FUNCTION_BLOCK GEOLOC_SUBSCRIBER_SINGLE
  {SET_ATTRIBUTE(OpcUa, SERVICE)}
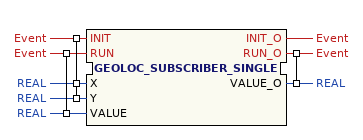
  EVENT_INPUT
    INIT WITH X, Y; (* FB Initialization *)
    RUN WITH VALUE; (* Read Event *)
  END_EVENT
  EVENT_OUTPUT
    INIT_O; (* Initialization Confirm *)
    RUN_O WITH VALUE_O; (* Read Event *)
  END_EVENT
  VAR_INPUT
    X : REAL; (* Latitude *)
    Y : REAL; (* Longitude *)
    VALUE : REAL; (* Read Value *)
  END_VAR
  VAR_OUTPUT
    VALUE_O : REAL; (* Read Value *)
  END_VAR
END_FUNCTION_BLOCK
